// TIA Portal V18 export
DATA_BLOCK "LEDS_DB"   // DB17
// stored: AutoNumber false, InstanceOfName LEDS, InstanceOfType FB
"LEDS"
   // VAR
   //    ElevClLEDStatus : Bool;
   //    MSVClLEDStatus : Bool;
   //    BUWClLEDStatus : Bool;
   // END_VAR
BEGIN
END_DATA_BLOCK
